PROGRAM prgComEffIO
VAR
	fbCom		: FB_MqttCommunicator_V3;
END_VAR

fbCom(
	bConnect				:= TRUE,
	strAuthKey				:= 'BMS99299754422' , 
	sUserName				:= 'c206f4dc-878b-4b9d-a673-4d85a4e99aa5', 
	sUserPassword			:= 'b59c3c46-e011-4210-beab-98c111b9c9fa', 
	eSavePositionCertificate:= eSavePositionOnPLC.ePostionHardDisk, 
	time_HeartBeat_sec := T#15S,
	bConnected=> , 
	bError=> , 
	hrErrorCode=> , 
	eConnectionState=> , 
	eErrorMessage_Out=> );

END_PROGRAM

(* stored: Version 1.1.0.1, ProductVersion 3.1.4024.12
   POU prgComEffIO: Id {cbcd318b-bf51-484c-bcaa-d6efcdf43fe3}, SpecialFunc None *)
